// TIA Portal V16 export
// export: Created 2022-07-21T09:35:24.3654793Z, ExportSetting WithDefaults, DisplayName Totally Integrated Automation Portal, DisplayVersion V16 Update 4, DisplayName TIA Portal Version Control Interface, DisplayVersion V16 Update 2, DisplayName TIA Portal Openness, DisplayVersion V16 Update 4, DisplayName SINAMICS Startdrive Advanced, DisplayVersion V16 Update 5, DisplayName SINAMICS Startdrive G130, G150, S120, S150, SINAMICS MV, S210, DisplayVersion V16 Update 5, DisplayName SINAMICS Startdrive G110M, G120, G120C, G120D, G120P, G115D, DisplayVersion V16 Update 5, DisplayName STEP 7 Professional, DisplayVersion V16 Update 4, DisplayName STEP 7 Safety, DisplayVersion V16, DisplayName WinCC Advanced, DisplayVersion V16 Update 4
FUNCTION "fcAnalogFestoSensor" : Void   // FC30, LAD
TITLE = Analog sensor (value from IO-Link) / Blok do obslugi czujnika analogowego (wartość z IO-Link)
{ S7_Optimized_Access := 'TRUE' }
VERSION : 0.1
// stored: AutoNumber true, IsIECCheckEnabled false, SetENOAutomatically false, UDAEnableTagReadback false
   VAR_INPUT
      inSensorMin : Real;
      inSensorMax : Real;
      inSensorValue : Word;
      inRangeMin : Real;
      inRangeMax : Real;
   END_VAR
   VAR_OUTPUT
      ouValue : Real;
      ouValueInRange : Bool;
   END_VAR
   VAR_TEMP
      tVacumNorm : Real;
      tVacumScale : Real;
      tVacumScaleABS : Real;
      tRangeMinABS : Real;
      tRangeMaxABS : Real;
   END_VAR
BEGIN

REGION Network 1: Pressure sensor value after scaling / Wartość z czujnika podciśnienia po przeskalowaniu
   // Najpierw normalizacja : 
   // Przeskalowanie wartości analogowej z zakresu 0 - 65532 (16#FFFC, wg. dokumentacji czujnika dwa pierwsze bity omijane) na zakres 0.0 - 1.0
   // 
   // Następnie skalowanie : 
   // Przeskalowanie zakresu 0.0 - 1.0 na zakres -1.0 +1.0 (wg dokumentacji z czujnika -1.0 do +1.0)
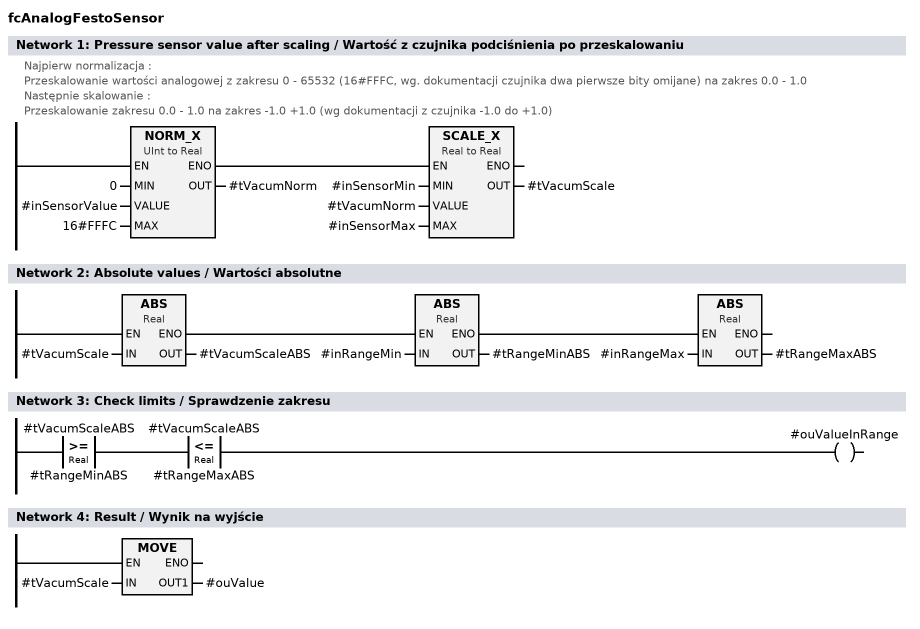
   RUNG wire#powerrail
      { S7_Templates := "[SrcType := UInt, DestType := Real]" } Normalize(min := 0, value := #inSensorValue, max := 16#FFFC, out => #tVacumNorm)
      { S7_Templates := "[SrcType := Real, DestType := Real]" } Scale(min := #inSensorMin, value := #tVacumNorm, max := #inSensorMax, out => #tVacumScale)
   END_RUNG
   // the same network as SCL:
   #tVacumNorm := NORM_X(MIN := 0, VALUE := #inSensorValue, MAX := 16#FFFC);
   #tVacumScale := SCALE_X(MIN := #inSensorMin, VALUE := #tVacumNorm, MAX := #inSensorMax);
END_REGION

REGION Network 2: Absolute values / Wartości absolutne
   RUNG wire#powerrail
      { S7_Templates := "SrcType := Real" } Abs(in := #tVacumScale, out => #tVacumScaleABS)
      { S7_Templates := "SrcType := Real" } Abs(in := #inRangeMin, out => #tRangeMinABS)
      { S7_Templates := "SrcType := Real" } Abs(in := #inRangeMax, out => #tRangeMaxABS)
   END_RUNG
   // the same network as SCL:
   #tVacumScaleABS := ABS(#tVacumScale);
   #tRangeMinABS := ABS(#inRangeMin);
   #tRangeMaxABS := ABS(#inRangeMax);
END_REGION

REGION Network 3: Check limits / Sprawdzenie zakresu
   RUNG wire#powerrail
      { S7_Templates := "SrcType := Real" } GE_Contact(in1 := #tVacumScaleABS, in2 := #tRangeMinABS)
      { S7_Templates := "SrcType := Real" } LE_Contact(in1 := #tVacumScaleABS, in2 := #tRangeMaxABS)
      Coil( #ouValueInRange )
   END_RUNG
   // the same network as SCL:
   #ouValueInRange := (#tVacumScaleABS >= #tRangeMinABS) AND (#tVacumScaleABS <= #tRangeMaxABS);
END_REGION

REGION Network 4: Result / Wynik na wyjście
   RUNG wire#powerrail
      Move(in := #tVacumScale, out1 => #ouValue)
   END_RUNG
   // the same network as SCL:
   #ouValue := #tVacumScale;
END_REGION
END_FUNCTION
